{attribute addProperty BoxType "EL6688-0000-0017"}
{attribute addProperty Id "External_SyncAT %I*External_Sync_AA57C188192240WcStateAT %I*WcState_98A4DF7520.250InfoDataAT %I*InfoData_0BDED7BF144180"}
{attribute addProperty CRC "3911825426"}
{attribute addProperty SizeInBites "338"}
{attribute addProperty SizeInBytes "42.25"}
TYPE EL6688_CA73E613 :
STRUCT
	{attribute addProperty Name "External_Sync"}
	External_Sync : External_Sync_AA57C188;
	{attribute addProperty Name "WcState"}
	WcState : WcState_98A4DF75;
	{attribute addProperty Name "InfoData"}
	InfoData : InfoData_0BDED7BF;
END_STRUCT
END_TYPE

(* stored: Version 1.2.0.0, ProductVersion 3.1.4024.9
   DUT EL6688_CA73E613: Id {a4e02c83-60cb-4d62-934a-2968237effda} *)
